// CASE: E_AlarmMessage.Insert
IF nStep = E_AlarmMessage.Insert THEN
	
	stEventEntryTemp.sSourceName := fbEvent.ipSourceInfo.sName;
	stEventEntryTemp.nSourceId := fbEvent.ipSourceInfo.nId;
	stEventEntryTemp.eSeverity := fbEvent.eSeverity;
	IF stEventEntryTemp.eSeverity = 0 THEN stEventEntryTemp.sSeverity := 'Verbose';
	ELSIF stEventEntryTemp.eSeverity = 1 THEN stEventEntryTemp.sSeverity := 'Info';
	ELSIF stEventEntryTemp.eSeverity = 2 THEN stEventEntryTemp.sSeverity := 'Warning';
	ELSIF stEventEntryTemp.eSeverity = 3 THEN stEventEntryTemp.sSeverity := 'Error';
	ELSIF stEventEntryTemp.eSeverity = 4 THEN stEventEntryTemp.sSeverity := 'Critical'; END_IF
	stEventEntryTemp.EventClass := fbEvent.EventClass;
	stEventEntryTemp.nEventId := fbEvent.nEventId;
	stEventEntryTemp.ipArguments := fbEvent.ipArguments;

	IF TestandSet(bEventEntryTableTestandSet) THEN

		nConfirmEntryIndex := GetIndex(stEventEntryTemp, FALSE);
		IF nConfirmEntryIndex >= 0 THEN
			aEventEntryTable[nConfirmEntryIndex].bLogged := FALSE;
			aEventEntryTable[nConfirmEntryIndex].eConfirmationState := TcEventConfirmationState.Confirmed;
			aEventEntryTable[nConfirmEntryIndex].sTimestampConfirmed := SYSTEMTIME_TO_STRING(UlintToSystemTime(fbEvent.nTimestamp, fbGetTimeZoneInformation.tzInfo));
			aEventEntryTable[nConfirmEntryIndex].sTimestampLog := aEventEntryTable[nConfirmEntryIndex].sTimestampConfirmed;
			stEventEntryTemp := aEventEntryTable[nConfirmEntryIndex];
			nCounterNothingFound := 0;
		ELSE
			nCounterNothingFound := nCounterNothingFound + 1;
			IF nCounterNothingFound <= 20 THEN 
				bEventEntryTableTestandSet := FALSE;
				RETURN;	
			END_IF
			nCounterNothingFound := 0;	
		END_IF

		stSeverestAlarmEntryTable := GetSeverestAlarmEntryTable();
		stLastEventEntryTable := GetLastEventEntryTable(); 
		UpdateLegacyTable();
	
		stEventEntryTemp.stAlarmLog.sTimestamp := stEventEntryTemp.sTimestampLog;      
		stEventEntryTemp.stAlarmLog.eConfirmationState := stEventEntryTemp.eConfirmationState;
		stEventEntryTemp.stAlarmLog.eSeverity := stEventEntryTemp.eSeverity;
		stEventEntryTemp.stAlarmLog.EventClassName := stEventEntryTemp.EventClassName;
		stEventEntryTemp.stAlarmLog.sSourceName := stEventEntryTemp.sSourceName;
		stEventEntryTemp.stAlarmLog.sText := stEventEntryTemp.sText;
		stEventEntryTemp.stAlarmLog.sTimestamp := REPLACE(STR1:= stEventEntryTemp.stAlarmLog.sTimestamp, STR2 := ' ',L := 1, P := 11);
	
		nStep := E_AlarmMessage.Done;
					
		bEventEntryTableTestandSet := FALSE;
	END_IF
END_IF

// CASE: Done   
IF nStep = E_AlarmMessage.Done THEN  
	OnAlarmConfirmed := S_OK;
	nStep := E_AlarmMessage.RequestText;
	MEMSET(destAddr := ADR(stEventEntryTemp), fillByte := 16#00 , n:= SIZEOF(stEventEntryTemp)); 
END_IF     

// Fast Case of nStepRequestText
// CASE: RequestText   
IF nStepRequestText = E_AlarmMessage.RequestText THEN
	fbRequestText.Request(eventClass:=fbEvent.EventClass, nEventId:=fbEvent.nEventId, nLangId:=LangId, ipArgs:=fbEvent.ipArguments );
	nStepRequestText := E_AlarmMessage.ReceiveText; 
END_IF
// CASE: ReceiveText   
IF nStepRequestText = E_AlarmMessage.ReceiveText THEN
	IF NOT fbRequestText.bBusy AND NOT fbRequestText.bError THEN
		fbRequestText.GetString(UTF8, SIZEOF(UTF8));
		UTF8_TO_STRING(pDstSTRING:=ADR(stEventEntryTemp.sText) , pSrcUTF8:=ADR(UTF8) , nDstSize:=SIZEOF(stEventEntryTemp.sText) , nDstLen=> );
		nStepRequestText := E_AlarmMessage.Done;
	ELSIF fbRequestText.bError THEN 
		nStepRequestText := E_AlarmMessage.RequestText;
	END_IF 
END_IF
 
// Fast Case of nStepRequestClass
// CASE: RequestText   
IF nStepRequestClass = E_AlarmMessage.RequestText THEN
	fbRequestClassName.Request(eventClass:=fbEvent.EventClass, nLangId:=LangId,);
	nStepRequestClass := E_AlarmMessage.ReceiveText;
END_IF
// CASE: ReceiveText   
IF nStepRequestClass = E_AlarmMessage.ReceiveText THEN
	IF NOT fbRequestClassName.bBusy AND NOT fbRequestClassName.bError THEN
		fbRequestClassName.GetString(UTF8, SIZEOF(UTF8));
		UTF8_TO_STRING(pDstSTRING:=ADR(stEventEntryTemp.EventClassName) , pSrcUTF8:=ADR(UTF8) , nDstSize:=SIZEOF(stEventEntryTemp.EventClassName) , nDstLen=> );
		nStepRequestClass := E_AlarmMessage.Done;
	ELSIF fbRequestClassName.bError THEN 
		nStepRequestClass := E_AlarmMessage.RequestText;
	END_IF
END_IF
END_METHOD

METHOD OnAlarmRaised : HRESULT
VAR_INPUT
	fbEvent : REFERENCE TO FB_TcEvent;
END_VAR
VAR
    hr : HRESULT;
    UTF8 : STRING(255);
END_VAR
VAR_INST
    {attribute 'no_copy'}
    fbRequestText : FB_RequestEventText;
    {attribute 'no_copy'}
    fbRequestClassName : FB_RequestEventClassName;
END_VAR
VAR_INST
    stEventEntryTemp: ST_EventEntryTableListener;
END_VAR
VAR_INST
    nStep : E_AlarmMessage;
    nStepRequestText : E_AlarmMessage := E_AlarmMessage.Done;
    nStepRequestClass : E_AlarmMessage := E_AlarmMessage.Done;
END_VAR

IF NOT __ISVALIDREF(fbEvent) THEN
	RETURN;
ELSE
	OnAlarmRaised := E_FAIL; // in order to receive more callbacks (Set <> S_OK in order to cancel the callbacks for this program cycle.)
	IF bChangeLanguageInterlock THEN
		RETURN;
	END_IF      
END_IF

// Fast Case of nStep
// CASE: E_AlarmMessage.RequestText
IF nStep = E_AlarmMessage.RequestText THEN
	nStepRequestText := E_AlarmMessage.RequestText;
	nStepRequestClass := E_AlarmMessage.RequestText;
	nStep := E_AlarmMessage.ReceiveText;
END_IF

// CASE: E_AlarmMessage.ReceiveText
IF nStep = E_AlarmMessage.ReceiveText THEN
	IF nStepRequestText = E_AlarmMessage.Done AND
	   nStepRequestClass = E_AlarmMessage.Done THEN
	   nStep := E_AlarmMessage.Insert;
	END_IF
END_IF

// CASE: E_AlarmMessage.Insert
IF nStep = E_AlarmMessage.Insert THEN

	hr := fbEvent.GetJsonAttribute(stEventEntryTemp.sJsonAttribute, SIZEOF(stEventEntryTemp.sJsonAttribute));
	stEventEntryTemp.sSourceName := fbEvent.ipSourceInfo.sName;
	stEventEntryTemp.nSourceId := fbEvent.ipSourceInfo.nId;
	stEventEntryTemp.eSeverity := fbEvent.eSeverity;
	IF stEventEntryTemp.eSeverity = 0 THEN stEventEntryTemp.sSeverity := 'Verbose';
	ELSIF stEventEntryTemp.eSeverity = 1 THEN stEventEntryTemp.sSeverity := 'Info';
	ELSIF stEventEntryTemp.eSeverity = 2 THEN stEventEntryTemp.sSeverity := 'Warning';
	ELSIF stEventEntryTemp.eSeverity = 3 THEN stEventEntryTemp.sSeverity := 'Error';
	ELSIF stEventEntryTemp.eSeverity = 4 THEN stEventEntryTemp.sSeverity := 'Critical'; END_IF
	stEventEntryTemp.EventClass := fbEvent.EventClass;
	stEventEntryTemp.sTimestamp := SYSTEMTIME_TO_STRING(UlintToSystemTime(fbEvent.nTimestamp, fbGetTimeZoneInformation.tzInfo));
	stEventEntryTemp.sTimestampLog := stEventEntryTemp.sTimestamp;
	stEventEntryTemp.nEventId := fbEvent.nEventId;
	stEventEntryTemp.ipArguments := fbEvent.ipArguments;
	stEventEntryTemp.eConfirmationState := TcEventConfirmationState.WaitForConfirmation;
	stEventEntryTemp.bIsAlarm := TRUE;

	stEventEntryTemp.stAlarmLog.sTimestamp := stEventEntryTemp.sTimestampLog;      
	stEventEntryTemp.stAlarmLog.eConfirmationState := stEventEntryTemp.eConfirmationState;
	stEventEntryTemp.stAlarmLog.eSeverity := stEventEntryTemp.eSeverity;
	stEventEntryTemp.stAlarmLog.EventClassName := stEventEntryTemp.EventClassName;
	stEventEntryTemp.stAlarmLog.sSourceName := stEventEntryTemp.sSourceName;
	stEventEntryTemp.stAlarmLog.sText := stEventEntryTemp.sText;
	stEventEntryTemp.stAlarmLog.sTimestamp := REPLACE(STR1:= stEventEntryTemp.stAlarmLog.sTimestamp, STR2 := ' ',L := 1, P := 11);
            
	IF TestandSet(bEventEntryTableTestandSet) THEN
		SUCCEEDED(Insert(stEventEntryTable := stEventEntryTemp));

		UpdateLegacyTable();

		nStep := E_AlarmMessage.Done;

		bEventEntryTableTestandSet := FALSE;
	END_IF
END_IF

// CASE: Done   
IF nStep = E_AlarmMessage.Done THEN
	OnAlarmRaised := S_OK;
	nStep := E_AlarmMessage.RequestText;
	MEMSET(destAddr:= ADR(stEventEntryTemp), fillByte := 16#00 , n:= SIZEOF(stEventEntryTemp)); 
END_IF     

// Fast Case of nStepRequestText
// CASE: RequestText   
IF nStepRequestText = E_AlarmMessage.RequestText THEN
	fbRequestText.Request(eventClass:=fbEvent.EventClass, nEventId:=fbEvent.nEventId, nLangId:=LangId, ipArgs:=fbEvent.ipArguments );
	nStepRequestText := E_AlarmMessage.ReceiveText; 
END_IF
// CASE: ReceiveText   
IF nStepRequestText = E_AlarmMessage.ReceiveText THEN
	IF NOT fbRequestText.bBusy AND NOT fbRequestText.bError THEN
		fbRequestText.GetString(UTF8, SIZEOF(UTF8));
		UTF8_TO_STRING(pDstSTRING:=ADR(stEventEntryTemp.sText) , pSrcUTF8:=ADR(UTF8) , nDstSize:=SIZEOF(stEventEntryTemp.sText) , nDstLen=> );
		nStepRequestText := E_AlarmMessage.Done;
	ELSIF fbRequestText.bError THEN 
		nStepRequestText := E_AlarmMessage.RequestText;
	END_IF 
END_IF
 
// Fast Case of nStepRequestClass
// CASE: RequestText   
IF nStepRequestClass = E_AlarmMessage.RequestText THEN
	fbRequestClassName.Request(eventClass:=fbEvent.EventClass, nLangId:=LangId,);
	nStepRequestClass := E_AlarmMessage.ReceiveText;
END_IF
// CASE: ReceiveText   
IF nStepRequestClass = E_AlarmMessage.ReceiveText THEN
	IF NOT fbRequestClassName.bBusy AND NOT fbRequestClassName.bError THEN
		fbRequestClassName.GetString(UTF8, SIZEOF(UTF8));
		UTF8_TO_STRING(pDstSTRING:=ADR(stEventEntryTemp.EventClassName) , pSrcUTF8:=ADR(UTF8) , nDstSize:=SIZEOF(stEventEntryTemp.EventClassName) , nDstLen=> );
		nStepRequestClass := E_AlarmMessage.Done;
	ELSIF fbRequestClassName.bError THEN 
		nStepRequestClass := E_AlarmMessage.RequestText;
	END_IF
END_IF
END_METHOD

METHOD OnMessageSent : HRESULT
VAR_INPUT
	fbEvent : REFERENCE TO FB_TcEvent;
END_VAR
VAR
    hr : HRESULT;
    UTF8 : STRING(255);
END_VAR
VAR_INST
    {attribute 'no_copy'}
    fbRequestText : FB_RequestEventText;
    {attribute 'no_copy'}
    fbRequestClassName : FB_RequestEventClassName;
END_VAR
VAR_INST
    stEventEntryTemp: ST_EventEntryTableListener;
END_VAR
VAR_INST
    nStep : E_AlarmMessage;
    nStepRequestText : E_AlarmMessage := E_AlarmMessage.Done;
    nStepRequestClass : E_AlarmMessage := E_AlarmMessage.Done;
END_VAR
VAR_INST
    nCyclesPerMessage : UINT;
END_VAR

IF NOT __ISVALIDREF(fbEvent) THEN
	RETURN;
ELSE
    OnMessageSent := E_FAIL;	// in order to receive more callbacks (Set <> S_OK in order to cancel the callbacks for this program cycle.)
    IF bChangeLanguageInterlock THEN
		RETURN;
    END_IF    
END_IF

// Fast Case of nStep
// CASE: E_AlarmMessage.RequestText
nCyclesPerMessage := nCyclesPerMessage + 1;
    IF nStep = E_AlarmMessage.RequestText THEN
        nStepRequestText := E_AlarmMessage.RequestText;
        nStepRequestClass := E_AlarmMessage.RequestText;
        nStep := E_AlarmMessage.ReceiveText;
	END_IF
    // CASE: E_AlarmMessage.ReceiveText
    IF nStep = E_AlarmMessage.ReceiveText THEN
        IF nStepRequestText = E_AlarmMessage.Done AND
           nStepRequestClass = E_AlarmMessage.Done THEN
           nStep := E_AlarmMessage.Insert;
		END_IF
	END_IF
    // CASE: E_AlarmMessage.Insert
    IF nStep = E_AlarmMessage.Insert THEN
        
            hr := fbEvent.GetJsonAttribute(stEventEntryTemp.sJsonAttribute, SIZEOF(stEventEntryTemp.sJsonAttribute));
            stEventEntryTemp.sSourceName := fbEvent.ipSourceInfo.sName;
            stEventEntryTemp.eSeverity := fbEvent.eSeverity;
            IF stEventEntryTemp.eSeverity = 0 THEN stEventEntryTemp.sSeverity := 'Verbose';
            ELSIF stEventEntryTemp.eSeverity = 1 THEN stEventEntryTemp.sSeverity := 'Info';
            ELSIF stEventEntryTemp.eSeverity = 2 THEN stEventEntryTemp.sSeverity := 'Warning';
            ELSIF stEventEntryTemp.eSeverity = 3 THEN stEventEntryTemp.sSeverity := 'Error';
            ELSIF stEventEntryTemp.eSeverity = 4 THEN stEventEntryTemp.sSeverity := 'Critical'; END_IF
            stEventEntryTemp.EventClass := fbEvent.EventClass;
            stEventEntryTemp.sTimestamp := SYSTEMTIME_TO_STRING(UlintToSystemTime(fbEvent.nTimestamp, fbGetTimeZoneInformation.tzInfo));
            stEventEntryTemp.sTimestampLog := stEventEntryTemp.sTimestamp;
            stEventEntryTemp.nEventId := fbEvent.nEventId;
            stEventEntryTemp.ipArguments := fbEvent.ipArguments;
            stEventEntryTemp.eConfirmationState := TcEventConfirmationState.NotRequired;
            stEventEntryTemp.bIsEvent := TRUE;
            
            stEventEntryTemp.stAlarmLog.sTimestamp := stEventEntryTemp.sTimestampLog;      
            stEventEntryTemp.stAlarmLog.eConfirmationState := stEventEntryTemp.eConfirmationState;
            stEventEntryTemp.stAlarmLog.eSeverity := stEventEntryTemp.eSeverity;
            stEventEntryTemp.stAlarmLog.EventClassName := stEventEntryTemp.EventClassName;
            stEventEntryTemp.stAlarmLog.sSourceName := stEventEntryTemp.sSourceName;
            stEventEntryTemp.stAlarmLog.sText := stEventEntryTemp.sText;
            stEventEntryTemp.stAlarmLog.sTimestamp := REPLACE(STR1:= stEventEntryTemp.stAlarmLog.sTimestamp, STR2 := ' ',L := 1, P := 11);
            
			IF TestandSet(bEventEntryTableTestandSet) THEN
            SUCCEEDED(Insert(stEventEntryTable := stEventEntryTemp));
                            
            UpdateLegacyTable();
            

            nStep := E_AlarmMessage.Done;

			bEventEntryTableTestandSet := FALSE;
			END_IF
	END_IF

    // CASE: Done   
    IF nStep = E_AlarmMessage.Done THEN
            OnMessageSent := S_OK;
            nStep := E_AlarmMessage.RequestText;
            MEMSET(destAddr:= ADR(stEventEntryTemp), fillByte := 16#00 , n:= SIZEOF(stEventEntryTemp)); 
	END_IF     


// Fast Case of nStepRequestText
    // CASE: RequestText   
    IF nStepRequestText = E_AlarmMessage.RequestText THEN
        fbRequestText.Request(eventClass:=fbEvent.EventClass, nEventId:=fbEvent.nEventId, nLangId:=LangId, ipArgs:=fbEvent.ipArguments );
        nStepRequestText := E_AlarmMessage.ReceiveText; 
	END_IF
    // CASE: ReceiveText   
    IF nStepRequestText = E_AlarmMessage.ReceiveText THEN
        IF NOT fbRequestText.bBusy AND NOT fbRequestText.bError THEN
            fbRequestText.GetString(UTF8, SIZEOF(UTF8));
            UTF8_TO_STRING(pDstSTRING:=ADR(stEventEntryTemp.sText) , pSrcUTF8:=ADR(UTF8) , nDstSize:=SIZEOF(stEventEntryTemp.sText) , nDstLen=> );
            nStepRequestText := E_AlarmMessage.Done;
        ELSIF fbRequestText.bError THEN 
            nStepRequestText := E_AlarmMessage.RequestText;
        END_IF 
	END_IF
 
// Fast Case of nStepRequestClass
    // CASE: RequestText   
    IF nStepRequestClass = E_AlarmMessage.RequestText THEN
        fbRequestClassName.Request(eventClass:=fbEvent.EventClass, nLangId:=LangId,);
        nStepRequestClass := E_AlarmMessage.ReceiveText;
	END_IF
    // CASE: ReceiveText   
    IF nStepRequestClass = E_AlarmMessage.ReceiveText THEN
        IF NOT fbRequestClassName.bBusy AND NOT fbRequestClassName.bError THEN
            fbRequestClassName.GetString(UTF8, SIZEOF(UTF8));
            UTF8_TO_STRING(pDstSTRING:=ADR(stEventEntryTemp.EventClassName) , pSrcUTF8:=ADR(UTF8) , nDstSize:=SIZEOF(stEventEntryTemp.EventClassName) , nDstLen=> );
            nStepRequestClass := E_AlarmMessage.Done;
        ELSIF fbRequestClassName.bError THEN 
            nStepRequestClass := E_AlarmMessage.RequestText;
        END_IF
	END_IF
END_METHOD

PROPERTY PUBLIC SeverestAlarmEntryTable : ST_EventEntryTableListener
GET
SeverestAlarmEntryTable := stSeverestAlarmEntryTable;
END_GET
END_PROPERTY

METHOD PRIVATE UlintToSystemTime : TIMESTRUCT
VAR_INPUT
	_fileTime: ULINT;
	_tzInfo: ST_TimeZoneInformation;
END_VAR
VAR
	tfileTime: T_FILETIME;
	tfileTimeZone: T_FILETIME;
	fbFileTimeToTzSpecificLocalTime: FB_FileTimeToTzSpecificLocalTime;
END_VAR
MEMCPY(ADR(tfileTime),ADR(_fileTime), SIZEOF(T_FILETIME));
fbFileTimeToTzSpecificLocalTime(
	in:= tfileTime, 
	tzInfo:= _tzInfo, 
	out=> tfileTimeZone, 
	eTzID=> , 
	bB=> );
UlintToSystemTime := FILETIME_TO_SYSTEMTIME(fileTime:= tfileTimeZone);
END_METHOD

METHOD PRIVATE UpdateLegacyTable : HRESULT
VAR
    i : DINT;
END_VAR
(* Class
0 None
1 Maintenance
2 Message
3 Hint
4 Information
5 Instruction
6 Warning
8 Parameter Error

Confirmation State
0 None
1 To Be Confirmed
2 None
3 Confirmation not needet
4 Confirmed
5 None

ResetState
0 None
1 RedExclamationMark
2 GreenFlag
3 Question Mark
4 None *)

FOR i := 1 TO TO_DINT(MIN(80,Parameter.nMaxEventEntries)) BY 1 DO

	// Severity
	CASE aEventEntryTable[i-1].eSeverity OF 
		TcEventSeverity.Verbose :
			aEvents[i].nClass := 0;
		TcEventSeverity.Info :
			aEvents[i].nClass := 4;
		TcEventSeverity.Warning :
			aEvents[i].nClass := 6; 
		TcEventSeverity.Error :
			aEvents[i].nClass := 7;
		TcEventSeverity.Critical :
			aEvents[i].nClass := 7;  
	END_CASE

	// state of confirmation and reset
	 CASE aEventEntryTable[i-1].eConfirmationState OF 
		TcEventConfirmationState.NotSupported :
			aEvents[i].nConfirmState := 0;
			aEvents[i].nResetState := 0;
			
		TcEventConfirmationState.NotRequired :
			aEvents[i].nConfirmState := 3;
			aEvents[i].nResetState := 0;
			
		TcEventConfirmationState.WaitForConfirmation :
			aEvents[i].nConfirmState := 1;
			aEvents[i].nResetState := 1;

		TcEventConfirmationState.Confirmed :
			aEvents[i].nConfirmState := 4;
			aEvents[i].nResetState := 3;
			
		TcEventConfirmationState.Reset :
			aEvents[i].nConfirmState := 0;
			aEvents[i].nResetState := 3;  
	END_CASE
  
	// rest of data
	aEvents[i].nEventId := aEventEntryTable[i-1].nEventId;
	aEvents[i].sComputer := aEventEntryTable[i-1].EventClassName;
	aEvents[i].sDate := LEFT( aEventEntryTable[i-1].sTimestamp, 10 );
	aEvents[i].sMessageText := aEventEntryTable[i-1].sText;
	aEvents[i].sSource := aEventEntryTable[i-1].sSourceName;
	aEvents[i].nSourceId := aEventEntryTable[i-1].nSourceId;
	aEvents[i].sTime := LEFT( DELETE( aEventEntryTable[i-1].sTimestamp, 11, 1 ), 8 );
	
 END_FOR
END_METHOD

END_FUNCTION_BLOCK

// ---- General/CONCAT/FB_CONCAT.TcPOU
FUNCTION_BLOCK FB_CONCAT 
VAR_INPUT
END_VAR
VAR_OUTPUT
END_VAR
VAR
    {attribute 'hide'}
	tmp:	STRING := '';
    {attribute 'hide'}
	_nDstSize	: UDINT;
	
	_fbConcatStrings	: FB_CONCAT_STRINGS;
END_VAR

METHOD PUBLIC SetDstString : I_CONCAT
VAR_INPUT
	anyDstString	: ANY_STRING;
END_VAR

_fbConcatStrings._pDstString := anyDstString.pValue;
_fbConcatStrings._nDstSize := DINT_TO_UDINT( anyDstString.diSize );
_fbConcatStrings._pDstString^ := '';

SetDstString := _fbConcatStrings;
END_METHOD

END_FUNCTION_BLOCK

// ---- General/CONCAT/FB_CONCAT_STRINGS.TcPOU
FUNCTION_BLOCK PUBLIC FB_CONCAT_STRINGS IMPLEMENTS I_CONCAT
VAR_INPUT
    {attribute 'hide'}
	_pDstString	: POINTER TO STRING;
    {attribute 'hide'}
	_nDstSize	: UDINT;
END_VAR
VAR_OUTPUT
END_VAR
VAR
END_VAR

// using a function like ADR() for input parameter gives no further recommendations in smart coding
METHOD PUBLIC AddString : I_CONCAT	// using a function like ADR() for input parameter gives no further recommendations in smart coding
VAR_INPUT
	pSrcString	: ANY_STRING;
END_VAR
CONCAT2(
	pSrcString1 := _pDstString,
	pSrcString2 := pSrcString.pValue,
	pDstString := _pDstString,
	nDstSize := _nDstSize
);
addString := THIS^;
END_METHOD

// Append text to the current build string.
METHOD PUBLIC AddStringInput : I_CONCAT
// comment below
VAR_INPUT
	in:	STRING;	// comment var
END_VAR

// comment implementation
addString( in );
addStringInput := THIS^;
END_METHOD

METHOD PUBLIC Get : T_MAXSTRING
VAR_INPUT
END_VAR

Get := _pDstString^;
END_METHOD

END_FUNCTION_BLOCK

// ---- EventLogger/Logger/FB_SystemTimeService.TcPOU
FUNCTION_BLOCK FB_SystemTimeService
VAR_INPUT
END_VAR
VAR_OUTPUT
END_VAR
VAR
    fbSystemTime    : FB_LocalSystemTime;
    sFileTimeString : STRING;
END_VAR


fbSystemTime(
	sNetID := '',
	bEnable := TRUE,
	dwCycle := 1,
	dwOpt := 0,
	tTimeout := DEFAULT_ADS_TIMEOUT
);

CalculateFileTimeString();

METHOD PRIVATE CalculateFileTimeString : BOOL
VAR_INPUT
END_VAR
VAR
    srawString      : STRING;
    sDeletedString  : STRING;
    sDeletedString2 : STRING;
END_VAR

srawString := ToString;

FindAndDeleteChar( ADR( srawString ), '-', ADR( sDeletedString ), SIZEOF( sDeletedString ) );
FindAndDeleteChar( ADR( sDeletedString ), ':', ADR( sDeletedString2 ), SIZEOF( sDeletedString2 ) );

sFileTimeSTring := Concat( Insert( LEFT( sDeletedString2, LEN( sDeletedString2 ) - 4 ), '_', 8 ), '_' );
END_METHOD

PROPERTY PUBLIC DateTime : DT
GET
DateTime := SYSTEMTIME_TO_DT( fbSystemTime.systemTime );
END_GET
END_PROPERTY

PROPERTY PUBLIC IsValid : BOOL
GET
IsValid := fbSystemTime.bValid;
END_GET
END_PROPERTY

PROPERTY PUBLIC TimeOfDay : TOD
GET
TimeOfDay := DT_TO_TOD( DateTime );
END_GET
END_PROPERTY

PROPERTY TimeOfDayToString : STRING
GET
TimeOfDayToString := RIGHT( ToString, 12 );
END_GET
END_PROPERTY

PROPERTY PUBLIC TimeStruct : REFERENCE TO TIMESTRUCT
GET
TimeStruct REF= fbSystemTime.systemTime;
END_GET
END_PROPERTY

PROPERTY PUBLIC ToFileTimeString : STRING
GET
ToFileTimeString := sFileTimeString;
END_GET
END_PROPERTY

PROPERTY ToString : STRING
GET
ToString := SYSTEMTIME_TO_STRING( fbSystemTime.systemTime );
END_GET
END_PROPERTY

END_FUNCTION_BLOCK

// ---- EventLogger/EventManagement/FB_AlarmDelayed.TcPOU
FUNCTION_BLOCK FB_AlarmDelayed EXTENDS FB_Alarm
VAR_INPUT
END_VAR
VAR_OUTPUT
END_VAR
VAR
	_tDelay		: TIME;
	_tonDelay	: TON;
END_VAR

METHOD FB_init : BOOL
VAR_INPUT
	bInitRetains : BOOL; // if TRUE, the retain variables are initialized (warm start / cold start)
	bInCopyCode : BOOL;  // if TRUE, the instance afterwards gets moved into the copy code (online change)
	
	stTmpEventClass	: TcEventEntry;
	tDelay			: TIME;
END_VAR

_tDelay := tDelay;
END_METHOD

// must be called cyclically once because of delay timer
METHOD PUBLIC setEvent : REFERENCE TO FB_Alarm
VAR_INPUT
	bSetEvent		: BOOL;	// cyclic call
END_VAR

_tonDelay(
	IN := bSetEvent,
	PT := _tDelay
);

SUPER^.setEvent( _tonDelay.Q );
setEvent REF= THIS^;
END_METHOD

// must be called cyclically once because of delay timer
METHOD PUBLIC setEventWithOneArgument : REFERENCE TO FB_Alarm
VAR_INPUT
	bSetEvent		: BOOL;	// cyclic call
	sInName			: STRING;
END_VAR
VAR_INST
	rtSetEvent		: R_TRIG;
END_VAR

_tonDelay(
	IN := bSetEvent,
	PT := _tDelay
);

SUPER^.setEventWithOneArgument( _tonDelay.Q, sInName );
setEventWithOneArgument REF= THIS^;
END_METHOD

END_FUNCTION_BLOCK

// ---- EventLogger/EventManagement/FB_Message.TcPOU
//Usage description
//-----------------
//| This FB uses the FB_init, which needs to be initialized within the declaration!
//| Also it can use the method Initialization, to specify Group/Zone IDs of the Event.
//| use Send( 0 ) send a message with current timestamp!
//| 
//| You can trigger an alarm once or use it cyclically.
//| The FB_ErrorManagement prevent acknowledge automatically if SetAlarm is still set.
FUNCTION_BLOCK FB_Message IMPLEMENTS I_Message
VAR_INPUT
END_VAR
VAR_OUTPUT
	sText		: STRING := '';
	sClassName	: STRING := '';
	sTimeRaised	: STRING := '';
	nGroupId	: UINT;
	nZoneId		: UINT;
END_VAR
VAR
	_bSetEvent				: BOOL;
	fbTcMessage				: FB_TcMessage;
//	_fbInternalSourceInfo	: Tc3_EventLogger.FB_TcSourceInfo;	// needed to have "multi-instances" of EventClass in CreateEx()
	nLangId					: INT;
	
    fbRequestText		: FB_RequestEventText;
    fbRequestClassName	: FB_RequestEventClassName;
	
	_stEventClass	: TcEventEntry;
	_nArgumentCount	: UDINT;
	
	hrRaise	: HRESULT;
END_VAR

METHOD Ack : HRESULT
VAR_INPUT
END_VAR

_bSetEvent := FALSE;
END_METHOD

METHOD PUBLIC AddArgument : REFERENCE TO FB_Message
VAR_INPUT
	sName	: STRING;
END_VAR

THIS^.fbTcMessage.ipArguments.AddString( sName );
addArgument REF= THIS^;
_nArgumentCount := _nArgumentCount + 1;
END_METHOD

PROPERTY PUBLIC bSetEvent : BOOL
GET
bSetEvent := _bSetEvent;
END_GET
SET
_bSetEvent := bSetEvent;
END_SET
END_PROPERTY

PROPERTY eSeverity : TcEventSeverity
GET
eSeverity := THIS^.fbTcMessage.eSeverity;
END_GET
END_PROPERTY

METHOD FB_init : BOOL
VAR_INPUT
	bInitRetains : BOOL; // if TRUE, the retain variables are initialized (warm start / cold start)
	bInCopyCode : BOOL;  // if TRUE, the instance afterwards gets moved into the copy code (online change)
	
	stTmpEventClass	: TcEventEntry;
END_VAR

// no online-change
IF NOT bInCopyCode THEN
	
	_stEventClass := stTmpEventClass;
	
	THIS^.fbTcMessage.CreateEx(
		_stEventClass,
		0
	);
		
END_IF
END_METHOD

METHOD GetEventEntry : ST_EventEntryTable
VAR_INPUT
END_VAR

GetEventEntry.sText := THIS^.sText;
GetEventEntry.sSourceName := THIS^.fbTcMessage.ipSourceInfo.sName;
GetEventEntry.nSourceId := THIS^.fbTcMessage.ipSourceInfo.nId;
GetEventEntry.nGroupId := THIS^.nGroupId;

GetEventEntry.sTimestamp := THIS^.sTimeRaised;

GetEventEntry.eSeverity := THIS^.fbTcMessage.eSeverity;
CASE THIS^.fbTcMessage.eSeverity OF
	TcEventSeverity.Verbose:	GetEventEntry.sSeverity := 'Verbose';
	TcEventSeverity.Info:		GetEventEntry.sSeverity := 'Info';
	TcEventSeverity.Warning:	GetEventEntry.sSeverity := 'Warning';
	TcEventSeverity.Error:		GetEventEntry.sSeverity := 'Error';
	TcEventSeverity.Critical:	GetEventEntry.sSeverity := 'Critical';
	ELSE	GetEventEntry.sSeverity := 'None';
END_CASE

GetEventEntry.EventClass := THIS^.fbTcMessage.EventClass;
GetEventEntry.EventClassName := THIS^.sClassName;

GetEventEntry.nEventId := THIS^.fbTcMessage.nEventId;
// GetEventEntry.ipArguments := fbTcAlarm.ipArguments;
GetEventEntry.bIsAlarm := TRUE;
GetEventEntry.bIsEvent := FALSE;

GetEventEntry.nLanguageId := THIS^.nLangId;

(*
	sJsonAttribute: STRING(8000);
#	sText: STRING(255); // 
#	sSourceName: STRING(255); // 
#	nSourceId: UDINT; // 
	sDescription: STRING(255);
#	eSeverity: TcEventSeverity; // INT
#	sSeverity: STRING;
#	EventClass: GUID;
#	EventClassName: STRING(255); //
	sTimestampLog : STRING;
	sTimestamp: STRING; // 
	sTimestampConfirmed: STRING;
	sTimestampCleared: STRING;
#	nEventId: UDINT;
#	ipArguments: I_TcArguments;
#	eConfirmationState: TcEventConfirmationState; // 
	bTextReceived: BOOL;
#	bIsAlarm: BOOL;
#	bIsEvent: BOOL;
	stAlarmLog : ST_AlarmLog;
	bLogged : BOOL;
#	nLanguageId : INT;
*)
END_METHOD

METHOD GetEventText : BOOL
VAR_INPUT
END_VAR
VAR_INST
	bReqTextError	: BOOL;
END_VAR

GetEventText := FALSE;

IF THIS^.fbTcMessage.RequestEventText(
	nLangId		:= 1031,
	sResult		:= sText,
	nResultSize	:= SIZEOF( sText ),
	bError		=> bReqTextError
) THEN
	GetEventText := TRUE;
END_IF

IF bReqTextError THEN
	sText := '';
END_IF
END_METHOD

METHOD GetJsonAttribute : HRESULT
VAR_INPUT
	sJsonAttribute	: REFERENCE TO STRING;
	nJsonAttribute	: UDINT;
END_VAR

THIS^.fbTcMessage.GetJsonAttribute( sJsonAttribute, nJsonAttribute );
END_METHOD

METHOD PUBLIC Initialize : HRESULT
VAR_INPUT
	nTmpZoneId			: UINT;
	nTmpGroupId			: UINT;
	eInEventReaction	: E_AlarmReaction;
END_VAR

THIS^.nZoneId := nTmpZoneId;
THIS^.nGroupId := nTmpGroupId;
END_METHOD

PROPERTY PUBLIC ipArguments : I_TcArguments
GET
ipArguments := THIS^.fbTcMessage.ipArguments;
END_GET
END_PROPERTY

PROPERTY PUBLIC LogEntry : ST_LogEntry
GET

LogEntry.sText := sText;
LogEntry.sTimestampLog := sTimeRaised;
LogEntry.sSeverity := THIS^.sSeverity;
LogEntry.sSourceName := THIS^.fbTcMessage.ipSourceInfo.sName;
END_GET
END_PROPERTY

PROPERTY PUBLIC nGetGroupId : UINT
GET
nGetGroupId := nGroupId;
END_GET
END_PROPERTY

PROPERTY PUBLIC nGetSourceId : UDINT
GET
nGetSourceId := THIS^.fbTcMessage.ipSourceInfo.nId;
END_GET
END_PROPERTY

METHOD PUBLIC SetEvent : REFERENCE TO FB_Message
VAR_INPUT
	bSetEvent	: BOOL;
END_VAR

IF bSetEvent
AND_THEN NOT THIS^._bSetEvent THEN
	hrRaise := THIS^.fbTcMessage.Send( 0 );
	GVL_Diag.gfbLogFile.addEntry( THIS^ );

THIS^.sTimeRaised := SYSTEMTIME_TO_STRING(
	UlintToSystemTime(
		THIS^.fbTcMessage.nTimeSent,
		GVL_Diag.gfbAlarmManagement.fbGetTimeZoneInformation.tzInfo ) );
		
END_IF
_bSetEvent := bSetEvent;

setEvent REF= THIS^;
END_METHOD

METHOD PUBLIC SetEventWithOneArgument : REFERENCE TO FB_Message
VAR_INPUT
	bSetEvent		: BOOL;	// cyclic call
	sInName			: STRING;
END_VAR
VAR_INST
	rtSetEvent		: R_TRIG;
END_VAR
VAR
    hr		: HRESULT;
    UTF8	: STRING(255);
END_VAR

IF bSetEvent
AND_THEN NOT THIS^._bSetEvent THEN
	THIS^.start().addArgument( sInName );
	hrRaise := THIS^.fbTcMessage.Send( 0 );
	GVL_Diag.gfbLogFile.addEntry( THIS^ );
END_IF
_bSetEvent := bSetEvent;

setEventWithOneArgument REF= THIS^;
END_METHOD

PROPERTY PRIVATE sSeverity : STRING
GET

CASE fbTcMessage.eSeverity OF
	
	TcEventSeverity.Critical:
		sSeverity := 'Critical';
		
	TcEventSeverity.Error:
		sSeverity := 'Error';
		
	TcEventSeverity.Info:
		sSeverity := 'Info';
		
	TcEventSeverity.Verbose:
		sSeverity := 'Verbose';
		
	TcEventSeverity.Warning:
		sSeverity := 'Warning';
		
	ELSE
		sSeverity := 'None';
		
END_CASE
END_GET
END_PROPERTY

METHOD PUBLIC Start : REFERENCE TO FB_Message
VAR_INPUT
END_VAR

THIS^.fbTcMessage.ipArguments.Clear();
start REF= THIS^;
_nArgumentCount := 0;
END_METHOD

METHOD PRIVATE UlintToSystemTime : TIMESTRUCT
VAR_INPUT
	_fileTime: ULINT;
	_tzInfo: ST_TimeZoneInformation;
END_VAR
VAR
	tfileTime: T_FILETIME;
	tfileTimeZone: T_FILETIME;
	fbFileTimeToTzSpecificLocalTime: FB_FileTimeToTzSpecificLocalTime;
END_VAR

MEMCPY( ADR( tfileTime ), ADR( _fileTime ), SIZEOF( T_FILETIME ) );
fbFileTimeToTzSpecificLocalTime(
	in := tfileTime, 
	tzInfo := _tzInfo, 
	out => tfileTimeZone, 
	eTzID => , 
	bB =>
);
UlintToSystemTime := FILETIME_TO_SYSTEMTIME( fileTime:= tfileTimeZone );
END_METHOD

END_FUNCTION_BLOCK

// ---- EventLogger/Logger/F_GetFileAgeInSeconds.TcPOU
FUNCTION F_GetFileAgeInSeconds : DINT
VAR_INPUT
    ActualTime    : T_FILETIME;
    FindFileEntry : ST_FindFileEntry;
END_VAR
VAR
    timeLastWriteAccess : T_ULARGE_INTEGER;
    fileTimeAsULINT     : T_ULARGE_INTEGER;
    fileTimeDifference  : T_ULARGE_INTEGER;
END_VAR


// Local file time
fileTimeAsULINT.dwLowPart := ActualTime.dwLowDateTime;
fileTimeAsULINT.dwHighPart := ActualTime.dwHighDateTime;

// Write access is UTC
timeLastWriteAccess.dwLowPart := FindFileEntry.lastWriteTime.dwLowDateTime;
timeLastWriteAccess.dwHighPart := FindFileEntry.lastWriteTime.dwHighDateTime;
fileTimeDifference := UInt64Sub64( fileTimeAsULINT, timeLastWriteAccess );

F_GetFileAgeInSeconds := LREAL_TO_DINT( UINT64_TO_LREAL( fileTimeDifference ) / ( 1000 * 1000 * 10 ) );

END_FUNCTION

// ---- General/Blinker/FB_Blinker.TcPOU
FUNCTION_BLOCK FB_Blinker
VAR_INPUT
	EN	: BOOL;	// enable
	PT	: TIME := T#500MS;
END_VAR
VAR_OUTPUT
	Q	: BOOL;
	Flash	: BOOL;	// flashes each rising edge of Q
END_VAR
VAR
	_tonBlink	: TON;
END_VAR

END_FUNCTION_BLOCK

// ---- General/Blinker/FB_Blinker_PWM.TcPOU
FUNCTION_BLOCK FB_Blinker_PWM
VAR_INPUT
	EN		: BOOL;	// enable
	PT		: TIME := T#500MS;
	PT_on	: TIME := T#250MS;
END_VAR
VAR_OUTPUT
	Q	: BOOL;
END_VAR
VAR
	_tonBlink	: TON;
	_tonPWM		: TON;
END_VAR


_tonBlink( IN := NOT _tonBlink.Q AND EN, PT := PT );
_tonPWM( IN := _tonBlink.IN, PT := PT_on );
Q := NOT _tonPWM.Q AND EN;

END_FUNCTION_BLOCK

// ---- General/FB_AnalogInputFilter.TcPOU
FUNCTION_BLOCK FB_AnalogInputFilter
VAR_INPUT
END_VAR
VAR_OUTPUT
	rVal:			LREAL := 0.0;	// Ausgangssignal
END_VAR
VAR
	rFactor:		LREAL;	// factor for filter
	rOldVal:		LREAL;	// old value to compare and calculate with
	bFirstCycle:	BOOL := TRUE;
END_VAR

METHOD FB_init : BOOL
VAR_INPUT
	bInitRetains : BOOL; // if TRUE, the retain variables are initialized (warm start / cold start)
	bInCopyCode : BOOL;  // if TRUE, the instance afterwards gets moved into the copy code (online change)
	
	rCycles		: REAL := 0.0;		// Anzahl Werte/Zyklen, über die 99% des Sollwerts erreicht werden soll.
END_VAR

// rCycles <= 0: pass-through (EXPT would explode at 1/0)
IF rCycles <= 0 THEN
	rFactor := 1;
ELSE
	// Faktor für die Gewichtung zwischen aktuellem und gespeicherten Wert
	// 0.01, da 1-0.99 wegen 99% als Ziel
	rFactor := 1 - LREAL_TO_REAL( EXPT(0.01, 1.0/rCycles) );
END_IF
END_METHOD

PROPERTY PUBLIC Value : LREAL
GET

Value := rVal;
END_GET
SET

// set value directly at first cycle to prevent startup ramp
IF bFirstCycle THEN
	rOldVal := Value;
	bFirstCycle := FALSE;
END_IF;

// filter value PT
rVal := (1 - rFactor) * rOldVal + rFactor * Value;
rOldVal := rVal;
END_SET
END_PROPERTY

END_FUNCTION_BLOCK

// ---- General/FB_Signal.TcPOU
FUNCTION_BLOCK FB_Signal
VAR_INPUT
	IN	: BOOL;	// state of signal
	PT_on	: TIME := T#200MS;
	PT_off	: TIME := T#200MS;
END_VAR
VAR_OUTPUT
	Q	: BOOL;	// effective value of signal
	Q_Stored	: BOOL;	// stored value of signal, reset manually with method
	RT	: BOOL;	// rising edge
	FT	: BOOL;	// falling edge
END_VAR
VAR
	tmpIN	: BOOL;
	
	tonOnDebounce	: TON;
	tofOffDebounce	: TOF;
END_VAR


// call timer to debounce signal
tonOnDebounce( IN := IN, PT := PT_on );
tofOffDebounce( IN := tonOnDebounce.Q, PT := PT_off );

Q := tofOffDebounce.Q;

// edges on debounced Q, not raw IN
RT := NOT tmpIN AND Q;
FT := tmpIN AND NOT Q;
Q_Stored S= Q;

// previous Q for next cycle
tmpIN := Q;

METHOD PUBLIC ResetQS : BOOL
VAR_INPUT
	reset	: BOOL;
END_VAR

IF reset THEN
	Q_Stored := FALSE;
END_IF
END_METHOD

END_FUNCTION_BLOCK

// ---- Lists/FB_ListNumbers_DINT.TcPOU
FUNCTION_BLOCK FB_ListNumbers_DINT
VAR_INPUT
END_VAR
VAR_OUTPUT
END_VAR
VAR
	i	: INT;
	asList	: ARRAY[0..MAX_INDEX] OF DINT;
END_VAR
VAR CONSTANT
	MAX_INDEX	: INT := 99;
END_VAR

METHOD PUBLIC AddEntry : BOOL
VAR_INPUT
	entry	: DINT;
END_VAR

AddEntry := FALSE;

// last slot occupied -> would drop data; refuse
IF asList[MAX_INDEX] <> 0 THEN
	RETURN;
END_IF

// shift elements in array
FOR i := MAX_INDEX - 1 TO 0 BY -1 DO
	asList[i+1] := asList[i];
END_FOR

asList[0] := entry;
AddEntry := TRUE;
END_METHOD

METHOD PUBLIC Clear : BOOL
VAR_INPUT
END_VAR

FOR i := 0 TO MAX_INDEX DO
	asList[i] := 0;
END_FOR
END_METHOD

METHOD PUBLIC PopEntry : DINT
VAR_INPUT
END_VAR

// return element
popEntry := asList[0];

// shift elements in array
FOR i := 0 TO MAX_INDEX - 1 DO
	asList[i] := asList[i + 1];
END_FOR
asList[MAX_INDEX] := 0;
END_METHOD

END_FUNCTION_BLOCK

// ---- Lists/FB_ListNumbers_REAL.TcPOU
FUNCTION_BLOCK FB_ListNumbers_REAL
VAR_INPUT
END_VAR
VAR_OUTPUT
END_VAR
VAR
	i	: INT;
	asList	: ARRAY[0..MAX_INDEX] OF REAL;
END_VAR
VAR CONSTANT
	MAX_INDEX	: INT := 99;
END_VAR

METHOD PUBLIC AddEntry : BOOL
VAR_INPUT
	entry	: REAL;
END_VAR

AddEntry := FALSE;

// last slot occupied -> would drop data; refuse
IF asList[MAX_INDEX] <> 0.0 THEN
	RETURN;
END_IF

// shift elements in array
FOR i := MAX_INDEX - 1 TO 0 BY -1 DO
	asList[i+1] := asList[i];
END_FOR

asList[0] := entry;
AddEntry := TRUE;
END_METHOD

METHOD PUBLIC Clear : BOOL
VAR_INPUT
END_VAR

FOR i := 0 TO MAX_INDEX DO
	asList[i] := 0;
END_FOR
END_METHOD

METHOD PUBLIC PopEntry : REAL
VAR_INPUT
END_VAR

// return element
popEntry := asList[0];

// shift elements in array
FOR i := 0 TO MAX_INDEX - 1 DO
	asList[i] := asList[i + 1];
END_FOR
asList[MAX_INDEX] := 0;
END_METHOD

END_FUNCTION_BLOCK

// ---- Lists/FB_ListString.TcPOU
FUNCTION_BLOCK FB_ListString
VAR_INPUT
END_VAR
VAR_OUTPUT
END_VAR
VAR
	asList	: ARRAY[0..MAX_INDEX] OF STRING;
END_VAR
VAR CONSTANT
	MAX_INDEX	: INT := 9;
END_VAR


// FIFO

METHOD addEntry : BOOL
VAR_INPUT
	entry	: STRING;
END_VAR
VAR
	i	: INT;
END_VAR

addEntry := FALSE;
FOR i := 0 TO MAX_INDEX DO
	IF asList[i] = '' THEN
		asList[i] := entry;
		addEntry := TRUE;
		EXIT;
	END_IF
END_FOR
END_METHOD

METHOD PUBLIC clear : BOOL
VAR_INPUT
END_VAR
VAR
	i	: INT;
END_VAR

FOR i := 0 TO MAX_INDEX DO
	asList[i] := '';
END_FOR
END_METHOD

METHOD PUBLIC isEmpty : BOOL
VAR_INPUT
END_VAR

isEmpty := asList[0] = '';
END_METHOD

METHOD PUBLIC popEntry : STRING
VAR_INPUT
END_VAR
VAR
	i	: INT;
END_VAR

// return element
popEntry := asList[0];

// shift elements in array
FOR i := 0 TO MAX_INDEX - 1 DO
	asList[i] := asList[i + 1];
END_FOR
asList[MAX_INDEX] := '';
END_METHOD

END_FUNCTION_BLOCK

// ---- Process/FB_Process.TcPOU
FUNCTION_BLOCK FB_Process
VAR_INPUT
END_VAR
VAR_OUTPUT
END_VAR
VAR
END_VAR

END_FUNCTION_BLOCK

// ---- Project Information/F_GetCompany.TcPOU
// This function has been automatically generated from the project information.
{attribute 'signature_flag' := '1073741824'}
{attribute 'TcGenerated'}
{attribute 'no-analysis'}
FUNCTION F_GetCompany : WSTRING
VAR_INPUT
	
END_VAR

F_GetCompany := "TwinCore";

END_FUNCTION

// ---- Project Information/F_GetTitle.TcPOU
// This function has been automatically generated from the project information.
{attribute 'signature_flag' := '1073741824'}
{attribute 'TcGenerated'}
{attribute 'no-analysis'}
FUNCTION F_GetTitle : WSTRING
VAR_INPUT
	
END_VAR

F_GetTitle := "TwinCore";

END_FUNCTION

// ---- Project Information/F_GetVersion.TcPOU
// This function has been automatically generated from the project information.
{attribute 'signature_flag' := '1073741824'}
{attribute 'TcGenerated'}
{attribute 'no-analysis'}
FUNCTION F_GetVersion : ST_LibVersion
VAR_INPUT
	
END_VAR

F_GetVersion.iMajor := 2026;
F_GetVersion.iMinor := 24;
F_GetVersion.iBuild := 1;
F_GetVersion.iRevision := 0;
F_GetVersion.sVersion := '2026.24.1.0';
F_GetVersion.nFlags := 1;

END_FUNCTION

// ---- StateMachine/MachineState/FB_MachineState.TcPOU
FUNCTION_BLOCK FB_MachineState
VAR_INPUT
	bInSwitchOn:			BOOL;	// switches on the machine
	bInSwitchOff:			BOOL;	// switches off the whole machine and screens
	bInMediaOn:				BOOL;	// switches on power, air pressure, etc.
	bInMediaOff:			BOOL;	// switches off power, air pressure, etc.
	bInStopCycleEnd:		BOOL;	// stop at the end of the current cycle
	bInReset:				BOOL;	// Reset / Acknowledge
	bInStart:				BOOL;	// Start automatic mode
	bInStop:				BOOL;	// Stops automatic mode immediately (manual control)
	
	
	bInHoming:				BOOL;	// war gelöscht, warum?
	bInClear:				BOOL;	// war gelöscht, warum?
	bInHold:				BOOL;	// war gelöscht, warum?
END_VAR
VAR_OUTPUT
	eMode:					E_Mode;
	bStateChanged:			BOOL;	// state has changed, TRUE for one cycle each state changing
	bStopAtCycleEndActive:	BOOL;
	
END_VAR
VAR
	fbMode:	FB_StateMachine;
	nMode:	E_Mode;
END_VAR


	CASE fbMode.nState OF

		E_Mode.Idle:
		
			fbMode.addStateCondition( bCondition := TRUE, sName:= 'Always TRUE' );
			
			IF fbMode.bStateChanged THEN
				;
			END_IF
			
			fbMode.addSwitchCondition( bCondition:= TRUE, sName:= 'Always TRUE' );
		
			IF fbMode.switch( sName:= 'Idle', tTimeout:= T#0S ) THEN
				fbMode.setNextState( E_Mode.Stopped );
			END_IF

		E_Mode.Homing:
		
			fbMode.addStateCondition( bCondition := TRUE, sName:= 'Always TRUE' );
			
			IF fbMode.bStateChanged THEN
				;
			END_IF
			
			fbMode.addSwitchCondition( bCondition:= TRUE, sName:= 'Always TRUE' );
		
			IF fbMode.switch( sName:= 'Homing', tTimeout:= T#0S ) THEN
				fbMode.setNextState( E_Mode.Starting );
			END_IF

		E_Mode.Starting:
		
			fbMode.addStateCondition( bCondition := TRUE, sName:= 'Always TRUE' );
			
			IF fbMode.bStateChanged THEN
				;
			END_IF
			
			fbMode.addSwitchCondition( bCondition:= TRUE, sName:= 'Always TRUE' );
		
			IF fbMode.switch( sName:= 'Starting', tTimeout:= T#0S ) THEN
				fbMode.setNextState( E_Mode.Execute );
			END_IF

		E_Mode.Hold:
		
			fbMode.addStateCondition( bCondition := TRUE, sName:= 'Always TRUE' );
			
			IF fbMode.bStateChanged THEN
				;
			END_IF
			
			fbMode.addSwitchCondition( bCondition:= TRUE, sName:= 'Always TRUE' );
		
			IF fbMode.switch( sName:= 'Execute', tTimeout:= T#0S ) THEN
				IF bInStart THEN	fbMode.setNextState( E_Mode.Execute ); END_IF
			END_IF

		E_Mode.Execute:
		
			fbMode.addStateCondition( bCondition := TRUE, sName:= 'Always TRUE' );
			
			IF fbMode.bStateChanged THEN
				;
			END_IF
			
			fbMode.addSwitchCondition( bCondition:= TRUE, sName:= 'Always TRUE' );
		
			IF fbMode.switch( sName:= 'Execute', tTimeout:= T#0S ) THEN
				fbMode.setNextState( E_Mode.Starting );
			END_IF
			IF bInHold THEN	fbMode.setNextState( E_Mode.Hold ); END_IF

		E_Mode.Stopping:
		
			fbMode.addStateCondition( bCondition := TRUE, sName:= 'Always TRUE' );
			
			IF fbMode.bStateChanged THEN
				;
			END_IF
			
			fbMode.addSwitchCondition( bCondition:= TRUE, sName:= 'Always TRUE' );
		
			IF fbMode.switch( sName:= 'Stopping', tTimeout:= T#0S ) THEN
				fbMode.setNextState( E_Mode.Stopped );
			END_IF

		E_Mode.Stopped:
		
			fbMode.addStateCondition( bCondition := TRUE, sName:= 'Always TRUE' );
			
			IF fbMode.bStateChanged THEN
				;
			END_IF
			
			fbMode.addSwitchCondition( bCondition := ( bInStart OR bInHoming OR bInClear ), sName := 'Clear, Home or Start' );
		
			IF fbMode.switch( sName:= 'Stopped', tTimeout:= T#0S ) THEN
				IF bInStart THEN	fbMode.setNextState( E_Mode.Starting ); END_IF
				IF bInHoming THEN	fbMode.setNextState( E_Mode.Homing ); END_IF
				IF bInClear THEN	fbMode.setNextState( E_Mode.Clearing ); END_IF
			END_IF

		E_Mode.Aborting:
		
			fbMode.addStateCondition( bCondition := TRUE, sName:= 'Always TRUE' );
			
			IF fbMode.bStateChanged THEN
				;
			END_IF
			
			fbMode.addSwitchCondition( bCondition:= TRUE, sName:= 'Always TRUE' );
		
			IF fbMode.switch( sName:= 'Aborting', tTimeout:= T#0S ) THEN
				fbMode.setNextState( E_Mode.Starting );
			END_IF

		E_Mode.Aborted:
			
			IF fbMode.bStateChanged THEN
				;
			END_IF
			
			fbMode.addSwitchCondition( bCondition:= bInClear, sName:= 'Acknowledge Error' );
		
			IF fbMode.switch( sName:= 'Aborted', tTimeout:= T#0S ) THEN
				fbMode.setNextState( E_Mode.Clearing );
			END_IF

		E_Mode.Clearing:
			
			IF fbMode.bStateChanged THEN
				;
			END_IF
			
			fbMode.addSwitchCondition( bCondition:= TRUE, sName:= 'Always TRUE' );
		
			IF fbMode.switch( sName:= 'Clearing', tTimeout:= T#0S ) THEN
				fbMode.setNextState( E_Mode.Stopped );
			END_IF

		E_Mode.Resetting:
		
			fbMode.addStateCondition( bCondition := TRUE, sName:= 'Always TRUE' );
			
			IF fbMode.bStateChanged THEN
				;
			END_IF
			
			fbMode.addSwitchCondition( bCondition:= TRUE, sName:= 'Always TRUE' );
		
			IF fbMode.switch( sName:= 'Resetting', tTimeout:= T#0S ) THEN
				fbMode.setNextState( E_Mode.Starting );
			END_IF
			
		E_Mode.Error:
			fbMode.setNextState( E_Mode.Aborted );
			
	END_CASE
	
	eMode := fbMode.nState;
	bStateChanged := fbMode.bStateChanged;

END_FUNCTION_BLOCK

// ---- StateMachine/ModeControl/FB_ModeControl.TcPOU
FUNCTION_BLOCK FB_ModeControl
VAR_INPUT
	bInAbort:				BOOL;
	bInHoming:				BOOL;
	bInHomePos:				BOOL;
	bInClear:				BOOL;
	bInReset:				BOOL;
	bInStart:				BOOL;
	bInHold:				BOOL;
	bInStop:				BOOL;
	bInStopCycleEnd:		BOOL;
	bInDone:				BOOL;	// state change possible
END_VAR
VAR_OUTPUT
	bOutLedStart:			BOOL;
	bOutLedStop:			BOOL;
	bOutLedHoming:			BOOL;
	bOutLedStopCycleEnd:	BOOL;
	eMode:					E_Mode;
	bStateChanged:			BOOL;	// state has changed, TRUE for one cycle each state changing
	bStopAtCycleEndActive:	BOOL;
	
END_VAR
VAR
	fbMode:	FB_StateMachine;
	nMode:	E_Mode;
END_VAR


	CASE fbMode.nState OF

		E_Mode.Idle:
		
			fbMode.addStateCondition( bCondition := TRUE, sName:= 'Always TRUE' );
			
			IF fbMode.bStateValid THEN
				;
			END_IF
			
			fbMode.addSwitchCondition( bCondition:= bInDone, sName:= 'not busy' );
		
			IF fbMode.switchWithDelay( sName:= 'Idle', tTimeout:= T#0S, tDelayTime := T#5s ) THEN
				fbMode.setNextState( E_Mode.Stopped );
			END_IF

		E_Mode.Homing:
		
			fbMode.addStateCondition( bCondition := TRUE, sName:= 'Always TRUE' );
			
			IF fbMode.bStateChanged THEN
				;
			END_IF
			
			fbMode.addSwitchCondition( bCondition:= bInDone, sName:= 'not busy' );
		
			IF fbMode.switch( sName:= 'Homing', tTimeout:= T#0S ) THEN
				fbMode.setNextState( E_Mode.Starting );
			END_IF

		E_Mode.Starting:
		
			fbMode.addStateCondition( bCondition := TRUE, sName:= 'Always TRUE' );
			
			IF fbMode.bStateChanged THEN
				;
			END_IF
			
			fbMode.addSwitchCondition( bCondition:= bInDone, sName:= 'not busy' );
		
			IF fbMode.switch( sName:= 'Starting', tTimeout:= T#0S ) THEN
				fbMode.setNextState( E_Mode.Execute );
			END_IF

		E_Mode.Hold:
		
			fbMode.addStateCondition( bCondition := TRUE, sName:= 'Always TRUE' );
			
			IF fbMode.bStateChanged THEN
				;
			END_IF
			
			fbMode.addSwitchCondition( bCondition:= bInDone, sName:= 'not busy' );
		
			IF fbMode.switch( sName:= 'Execute', tTimeout:= T#0S ) THEN
				IF bInStart THEN	fbMode.setNextState( E_Mode.Execute ); END_IF
			END_IF

		E_Mode.Standby:
		
			fbMode.addStateCondition( bCondition := TRUE, sName:= 'Always TRUE' );
			
			IF fbMode.bStateChanged THEN
				;
			END_IF
			
			fbMode.addSwitchCondition( bCondition:= bInStart OR bInStop, sName:= 'Start oder Stop' );
		
			IF fbMode.switch( sName:= 'Execute', tTimeout:= T#0S ) THEN
				IF bInStart THEN	fbMode.setNextState( E_Mode.Execute ); END_IF
				IF bInStop THEN	fbMode.setNextState( E_Mode.Stopping ); END_IF
				bInStart := bInStop := FALSE;
			END_IF

		E_Mode.Execute:
		
			fbMode.addStateCondition( bCondition := TRUE, sName:= 'Always TRUE' );
			
			IF fbMode.bStateChanged THEN
				;
			END_IF
			
			fbMode.addSwitchCondition( bCondition:= bInDone, sName:= 'not busy' );
		
			IF fbMode.switchWithDelay( sName:= 'Execute', tTimeout:= T#0S, tDelayTime := T#5S ) THEN
				fbMode.setNextState( E_Mode.Standby );
			END_IF
			IF bInHold THEN	fbMode.setNextState( E_Mode.Hold ); END_IF

		E_Mode.Stopping:
		
			fbMode.addStateCondition( bCondition := TRUE, sName:= 'Always TRUE' );
			
			IF fbMode.bStateChanged THEN
				;
			END_IF
			
			fbMode.addSwitchCondition( bCondition:= bInDone, sName:= 'not busy' );
		
			IF fbMode.switch( sName:= 'Stopping', tTimeout:= T#0S ) THEN
				fbMode.setNextState( E_Mode.Stopped );
			END_IF

		E_Mode.Stopped:
		
			fbMode.addStateCondition( bCondition := TRUE, sName:= 'Always TRUE' );
			
			IF fbMode.bStateChanged THEN
				;
			END_IF
			
			fbMode.addSwitchCondition( bCondition:= bInStart OR bInHoming OR bInClear, sName:= 'Clear, Home or Start' );
			fbMode.addSwitchCondition( bCondition:= bInDone, sName:= 'not busy' );
		
			IF fbMode.switch( sName:= 'Stopped', tTimeout:= T#0S ) THEN
				IF bInStart THEN	fbMode.setNextState( E_Mode.Starting ); END_IF
				IF bInHoming THEN	fbMode.setNextState( E_Mode.Homing ); END_IF
				IF bInClear THEN	fbMode.setNextState( E_Mode.Clearing ); END_IF
			END_IF

		E_Mode.Aborting:
		
			fbMode.addStateCondition( bCondition := TRUE, sName:= 'Always TRUE' );
			
			IF fbMode.bStateChanged THEN
				;
			END_IF
			
			fbMode.addSwitchCondition( bCondition:= bInDone, sName:= 'not busy' );
		
			IF fbMode.switch( sName:= 'Aborting', tTimeout:= T#0S ) THEN
				fbMode.setNextState( E_Mode.Starting );
			END_IF

		E_Mode.Aborted:
			
			IF fbMode.bStateChanged THEN
				;
			END_IF
			
			fbMode.addSwitchCondition( bCondition:= bInClear, sName:= 'Acknowledge Error' );
			fbMode.addSwitchCondition( bCondition:= bInDone, sName:= 'not busy' );
		
			IF fbMode.switch( sName:= 'Aborted', tTimeout:= T#0S ) THEN
				fbMode.setNextState( E_Mode.Clearing );
			END_IF

		E_Mode.Clearing:
			
			IF fbMode.bStateChanged THEN
				;
			END_IF
			
			fbMode.addSwitchCondition( bCondition:= bInDone, sName:= 'not busy' );
		
			IF fbMode.switch( sName:= 'Clearing', tTimeout:= T#0S ) THEN
				fbMode.setNextState( E_Mode.Stopped );
			END_IF

		E_Mode.Resetting:
		
			fbMode.addStateCondition( bCondition := TRUE, sName:= 'Always TRUE' );
			
			IF fbMode.bStateChanged THEN
				;
			END_IF
			
			fbMode.addSwitchCondition( bCondition:= bInDone, sName:= 'not busy' );
		
			IF fbMode.switch( sName:= 'Resetting', tTimeout:= T#0S ) THEN
				fbMode.setNextState( E_Mode.Starting );
			END_IF
			
		E_Mode.Error:
		
			fbMode.setNextState( E_Mode.Aborted );
			
	END_CASE
	
	eMode := fbMode.nState;
	bStateChanged := fbMode.bStateChanged;
	
	// Lamps
	bOutLedStart := fbMode.nState = E_Mode.Execute;
	bOutLedStop := fbMode.nState = E_Mode.Stopped;
	bOutLedHoming := bInHomePos;

END_FUNCTION_BLOCK
